// TIA Portal V17 export
// export: Created 2024-09-02T12:50:20.7933181Z, ExportSetting WithDefaults, DisplayName Totally Integrated Automation Portal, DisplayVersion V17, DisplayName TIA Portal Openness, DisplayVersion V17, DisplayName TIA Portal Version Control Interface, DisplayVersion V17, DisplayName STEP 7 Professional, DisplayVersion V17, DisplayName STEP 7 Safety, DisplayVersion V17, DisplayName WinCC Professional, DisplayVersion V17
DATA_BLOCK "MdsDB8_FG02_Status_Of_Communication_SLG3_OP70"   // DB1118
{ S7_Optimized_Access := 'TRUE'; DB_Accessible_From_OPC_UA := 'FALSE' }
AUTHOR : OlegFuehrus
FAMILY : MOBY
NAME : MOBY
VERSION : 0.1
// stored: AutoNumber false, DBAccessibleFromOPCUA false, IsOnlyStoredInLoadMemory false, IsRetainMemResEnabled false, IsWriteProtectedInAS false, MemoryReserve 100
   VAR
      Station : Struct   // Daten für Station / Data for station
         READING_START : Bool;   // Moby Lesen Start / Moby Read Start
         READING_FINISHED : Bool;   // Moby Lesen Fertig / moby read finished
         READING_START_FIXED : Bool;   // Moby Lesen Start Festbereich / Moby read start fixed area
         READING_FINISHED_FIXED : Bool;   // Moby Lesen Fertig Festbereich / Moby read finished fixed range
         READING_START_FLEX : Bool;   // Moby Lesen Start Flexibelbereich / Moby read start fixed area
         READING_FINISHED_FLEX : Bool;   // Moby Lesen Fertig Flexibelbereich / Moby finished flexible area
         WRITING_START : Bool;   // Moby Schreiben Start / Moby write done
         WRITING_FINISHED : Bool;   // Moby Schreiben Fertig / Moby write done
      END_STRUCT;
      ASM : Struct
         ERROR : Bool;   // Fehler Kommunikation SLG / Communication error SLG
         MDS_PRESENT : Bool;   // Datenträger anwesend / Data carrier present
         SYS : Struct   // System
            READING_START : Array[1..128] of Bool;
            READING_FINISHED : Array[1..128] of Bool;
            WRITING_START : Array[1..128] of Bool;
            WRITING_FINISHED : Array[1..128] of Bool;
         END_STRUCT;
         Free_Order : Struct   // Freier Auftrag / Free order
            READING_START : Array[1..6] of Bool;
            READING_FINISHED : Array[1..6] of Bool;
            WRITING_START : Array[1..6] of Bool;
            WRITING_FINISHED : Array[1..6] of Bool;
         END_STRUCT;
         INTERNALLY : Struct   // Intern / Internal
            READING_START : Array[1..8] of Bool;
            READING_FINISHED : Array[1..8] of Bool;
            WRITING_START : Array[1..8] of Bool;
            WRITING_FINISHED : Array[1..8] of Bool;
         END_STRUCT;
      END_STRUCT;
      Orders { S7_SetPoint := 'True'} : "TypeMobyBefehle";
      HMIDiag { S7_SetPoint := 'True'} : "TypeMobyHMIDiag";
   END_VAR
BEGIN
END_DATA_BLOCK
